// TIA Portal V15.1 export
// export: Created 2020-06-12T07:35:45.1318359Z, ExportSetting None, DisplayName Totally Integrated Automation Portal, DisplayVersion V15.1, DisplayName TIA Portal Openness, DisplayVersion V15.1, DisplayName STEP 7 Professional, DisplayVersion V15.1, DisplayName STEP 7 Safety, DisplayVersion V15.1, DisplayName WinCC Advanced, DisplayVersion V15.1
DATA_BLOCK "O2_DB"   // DB628
{ S7_Optimized_Access := 'TRUE' }
// stored: MemoryReserve 100
   VAR
      request : Int := 0;
      status { ExternalWritable := 'False'} : Word := 16#0000;
      air_on { ExternalAccessible := 'False'; ExternalVisible := 'False'; ExternalWritable := 'False'} : Bool := FALSE;
      o2_on { ExternalAccessible := 'False'; ExternalVisible := 'False'; ExternalWritable := 'False'} : Bool := FALSE;
      n2_on { ExternalAccessible := 'False'; ExternalVisible := 'False'; ExternalWritable := 'False'} : Bool := FALSE;
      clean_on { ExternalAccessible := 'False'; ExternalVisible := 'False'; ExternalWritable := 'False'} : Bool := FALSE;
      alm_en { ExternalAccessible := 'False'; ExternalVisible := 'False'; ExternalWritable := 'False'} : Bool := FALSE;   // Enable alarm
   END_VAR
   VAR RETAIN
      clean_count { ExternalWritable := 'False'} : Int := 0;
   END_VAR
   VAR
      action { ExternalAccessible := 'False'; ExternalVisible := 'False'; ExternalWritable := 'False'} : Int := 0;
   END_VAR
BEGIN
END_DATA_BLOCK
